FUNCTION_BLOCK Q_ChangeObjectLabel (* Command Change Object Label( Part 6 - F.50 ) *)
  (* Standard: ISO 11783-6; Description: Copyright (c) 2022 HR Agrartechnik GmbH This program and the accompanying materials are made available under the terms of the Eclipse Public License 2.0 which is available at https://www.eclipse.org/legal/epl-2.0/ SPDX-License-Identifier: EPL-2.0 see Description Tab *)
  (* Version 1.0, 2022-07-08, Franz Höpfinger, HR Agrartechnik GmbH *)
  (* Documentation:
  Command change background colour ( Part 6 - F.20 )
   This command is used to change the background colour of an object.
   param[in] {objectID, uint16_t}
   Object ID of object to associate label with
   param[in] {labelStringObjectID, uint16_t}
   Object ID of a String Variable object that contains the label string (32 characters maximum) or FFFF if no text is supplied
   param[in] {fontType, uint8_t}
   Font type (ignored if String Variable object reference is NULL or the string contains a WideString)
   param[in] {graphicalDesignatorObjectID, uint16_t}
   Object ID of an object to be used as a graphic representation of the object label or FFFF16 if no designator supplied.
   Return Values: 
   int16_t
    - VT_E_NO_ERR (0) - OK
   - VT_E_OVERFLOW (-6) - buffer overflow
   - VT_E_NOACT (-8) - Command not possible in current state
   - VT_E_NO_INSTANCE (-21) - No VT client available
   - VT_E_ISO_INSTANCE_INVALID (-129) - Identifier for instance (connection) invalid
   - VT_E_NOT_ALIVE (-130) - Identifier for instance valid, but VT Dead.
  *)
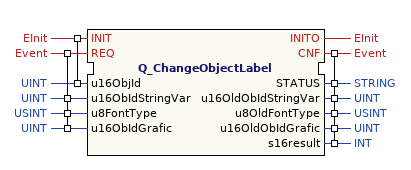
  EVENT_INPUT
    INIT : EInit WITH u16ObjId; (* Service Initialization *)
    REQ WITH u16ObIdStringVar, u8FontType, u16ObIdGrafic; (* Service Request *)
  END_EVENT
  EVENT_OUTPUT
    INITO : EInit; (* Initialization Confirm *)
    CNF WITH STATUS, u16OldObIdStringVar, u8OldFontType, u16OldObIdGrafic, s16result, u16OldObIdStringVar, u8OldFontType, u16OldObIdGrafic; (* Confirmation of Requested Service *)
  END_EVENT
  VAR_INPUT
    u16ObjId : UINT; (* Object ID *)
    u16ObIdStringVar : UINT; (* Object ID of a String Variable object that contains the label string (32 characters maximum) or FFFF if no text is supplied *)
    u8FontType : USINT; (* Font type (ignored if String Variable object reference is NULL or the string contains a WideString ) *)
    u16ObIdGrafic : UINT; (* Object ID of an object to be used as a graphic representation of the object label or FFFF16 if no designator supplied *)
  END_VAR
  VAR_OUTPUT
    STATUS : STRING; (* Service Status *)
    u16OldObIdStringVar : UINT; (* Old Object ID of a String Variable object that contains the label string (32 characters maximum) or FFFF if no text is supplied *)
    u8OldFontType : USINT; (* Old value for attribute *)
    u16OldObIdGrafic : UINT;
    s16result : INT; (* retval see description *)
  END_VAR
END_FUNCTION_BLOCK
